Fanuc KAREL source: kb00128.KL

-- PROVISIONAL review KL for V1013-1; original PC SHA256 85d1e9ea4e7407475a67ba307e2bfe235559bfcfa5e2166a3c8a3ceed80313ef
-- Incomplete behavior may be omitted. Consult companion uncertainty JSON. Do not deploy.
PROGRAM KB00128
%NOLOCKGROUP
BEGIN
  -- UNRESOLVED_PC offsets 5-28; opcodes 27,22,1C,31,4A
  -- UNRESOLVED_PC offsets 33-37; opcodes 7F
END KB00128
